(* Schneider Machine Expert - Basic project Modelo final v1.0, file version 2.5.0.0 *)
(* ProjectInformations: Name=Nuevo proyecto *)

HARDWARE
  Cpu 0: TM221CE24T
  EthernetConfiguration: NetworkName=M221, IpAllocationMode=FixedAddress, IpAddress=0.0.0.0, SubnetMask=0.0.0.0
  SerialLineConfiguration: Baud=Baud19200, Parity=ParityEven, DataBits=DataBits8, StopBits=StopBits1, PhysicalMedium=PhysicalMediumRs485, TransmissionMode=TransmissionModeModbusRtu, SlaveId=1, Addressing=SlaveAddressing
  MastTask: UsePeriodScanMode=false, PeriodScan=100
  FastTask: Period=255
  CpuBehavior: StartingMode=StartAsPreviousState, AutoSaveRamOnEeprom=true, WatchdogPeriod=250

SYMBOLS  (address, symbol, comment, settings)
  %M0         "Escalon frontal izquierdo"
  %M1         "Escalon frontal derecho"
  %M2         "Escalon trasero izquierdo"
  %M3         "Escalon trasero derecho"
  %M4         "Sensor frente izquierdo"
  %M5         "Sensor frente medio"
  %M6         "Sensor frente derecho"
  %M7         "Sensor derecha adelante"
  %M8         "Sensor derecha medio"
  %M9         "Sensor derecha atras"
  %M10        "Sensor trasero derecha"
  %M11        "Sensor trasero medio"
  %M12        "Sensor trasero izquierda"
  %M13        "Sensor izquierda atras"
  %M14        "Sensor izquierda medio"
  %M15        "Sensor izquierda adelante"
  %M40        "Reset gen"
  %S6       SB_TB1S  "Base de tiempo de 1 s generada por un reloj interno"
  %TM0        [Preset=5, Base=OneHundredMilliSeconds]
  %TM1        [Preset=5, Base=OneHundredMilliSeconds]
  %TM2        [Preset=5, Base=OneHundredMilliSeconds]
  %TM3        [Preset=5, Base=OneHundredMilliSeconds]
  %TM4        [Preset=5, Base=OneHundredMilliSeconds]
  %TM5        [Preset=5, Base=OneHundredMilliSeconds]
  %TM6        [Preset=5, Base=OneHundredMilliSeconds]
  %TM7        [Preset=5, Base=OneHundredMilliSeconds]
  %TM8        [Preset=5, Base=OneHundredMilliSeconds]
  %TM9        [Preset=5, Base=OneHundredMilliSeconds]
  %TM10       [Preset=5, Base=OneHundredMilliSeconds]
  %TM11       [Preset=5, Base=OneHundredMilliSeconds]
  %TM12       [Preset=5, Base=OneHundredMilliSeconds]
  %TM13       [Preset=5, Base=OneHundredMilliSeconds]
  %TM14       [Preset=5, Base=OneHundredMilliSeconds]
  %TM15       [Preset=5, Base=OneHundredMilliSeconds]
  %C0         [Preset=17]
  %I0.0     ENC1A  "Input"
  %I0.1     ENC1B  "Enable"
  %I0.6     ENC2A
  %I0.7     ENC2B
  %I0.8     MUX  "Data de mux sensores"
  %Q0.4     S0
  %Q0.5     S1
  %Q0.6     S2
  %Q0.7     S3

POU Demux
  (* SectionNumber=1 *)

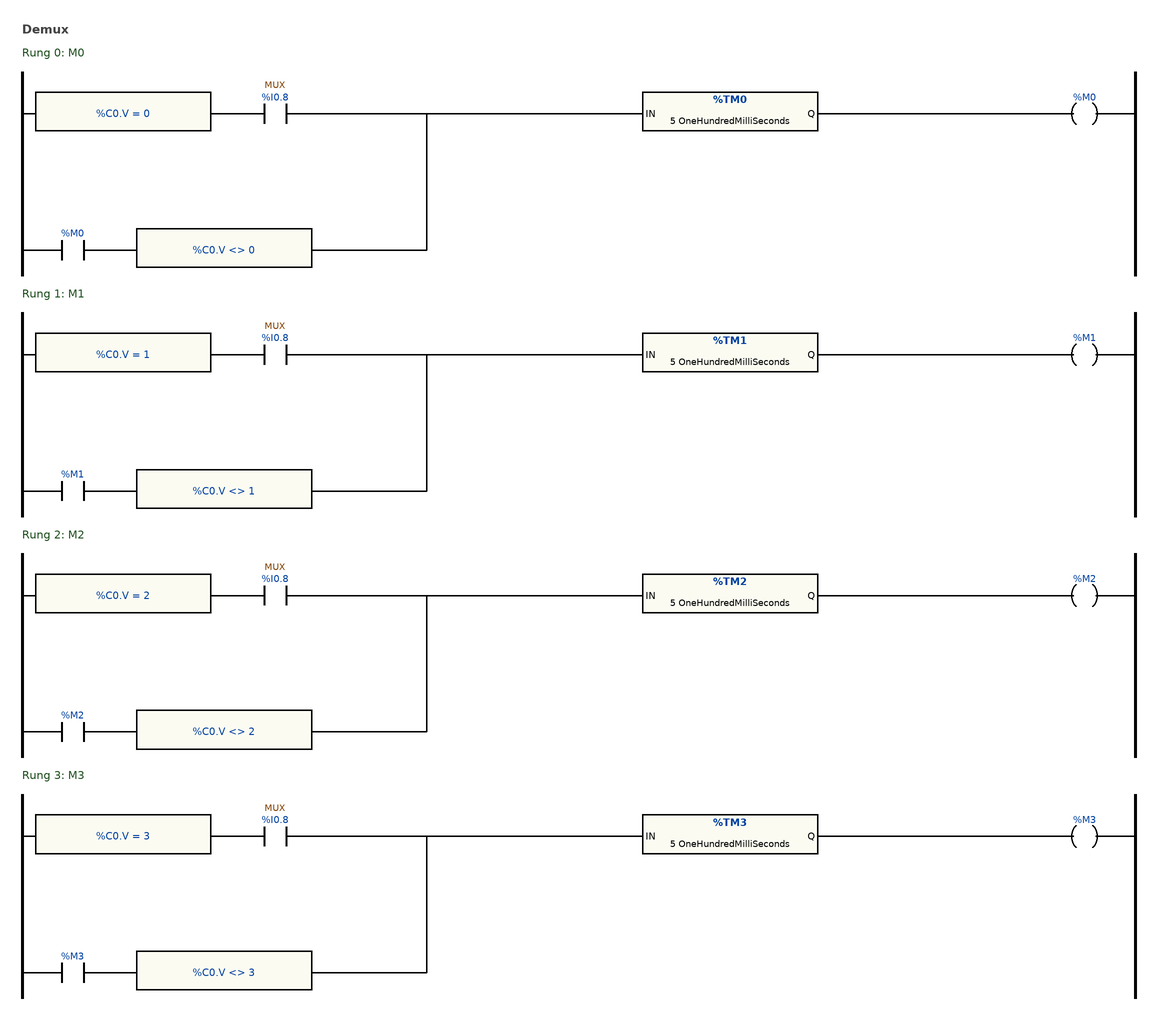

// Rung 0: M0
  BLK %TM0
  LD [ %C0.V = 0 ]
  AND %I0.8               (* MUX *)
  OR( %M0
  AND [ %C0.V <> 0 ]
  )
  IN
  OUT_BLK
  LD Q
  ST %M0
  END_BLK
  // as ST:
  //   %TM0(IN := %C0.V = 0 AND MUX OR %M0 AND %C0.V <> 0);
  //   %M0 := %TM0.Q;

// Rung 1: M1
  BLK %TM1
  LD [ %C0.V = 1 ]
  AND %I0.8               (* MUX *)
  OR( %M1
  AND [ %C0.V <> 1 ]
  )
  IN
  OUT_BLK
  LD Q
  ST %M1
  END_BLK
  // as ST:
  //   %TM1(IN := %C0.V = 1 AND MUX OR %M1 AND %C0.V <> 1);
  //   %M1 := %TM1.Q;

// Rung 2: M2
  BLK %TM2
  LD [ %C0.V = 2 ]
  AND %I0.8               (* MUX *)
  OR( %M2
  AND [ %C0.V <> 2 ]
  )
  IN
  OUT_BLK
  LD Q
  ST %M2
  END_BLK
  // as ST:
  //   %TM2(IN := %C0.V = 2 AND MUX OR %M2 AND %C0.V <> 2);
  //   %M2 := %TM2.Q;

// Rung 3: M3
  BLK %TM3
  LD [ %C0.V = 3 ]
  AND %I0.8               (* MUX *)
  OR( %M3
  AND [ %C0.V <> 3 ]
  )
  IN
  OUT_BLK
  LD Q
  ST %M3
  END_BLK
  // as ST:
  //   %TM3(IN := %C0.V = 3 AND MUX OR %M3 AND %C0.V <> 3);
  //   %M3 := %TM3.Q;

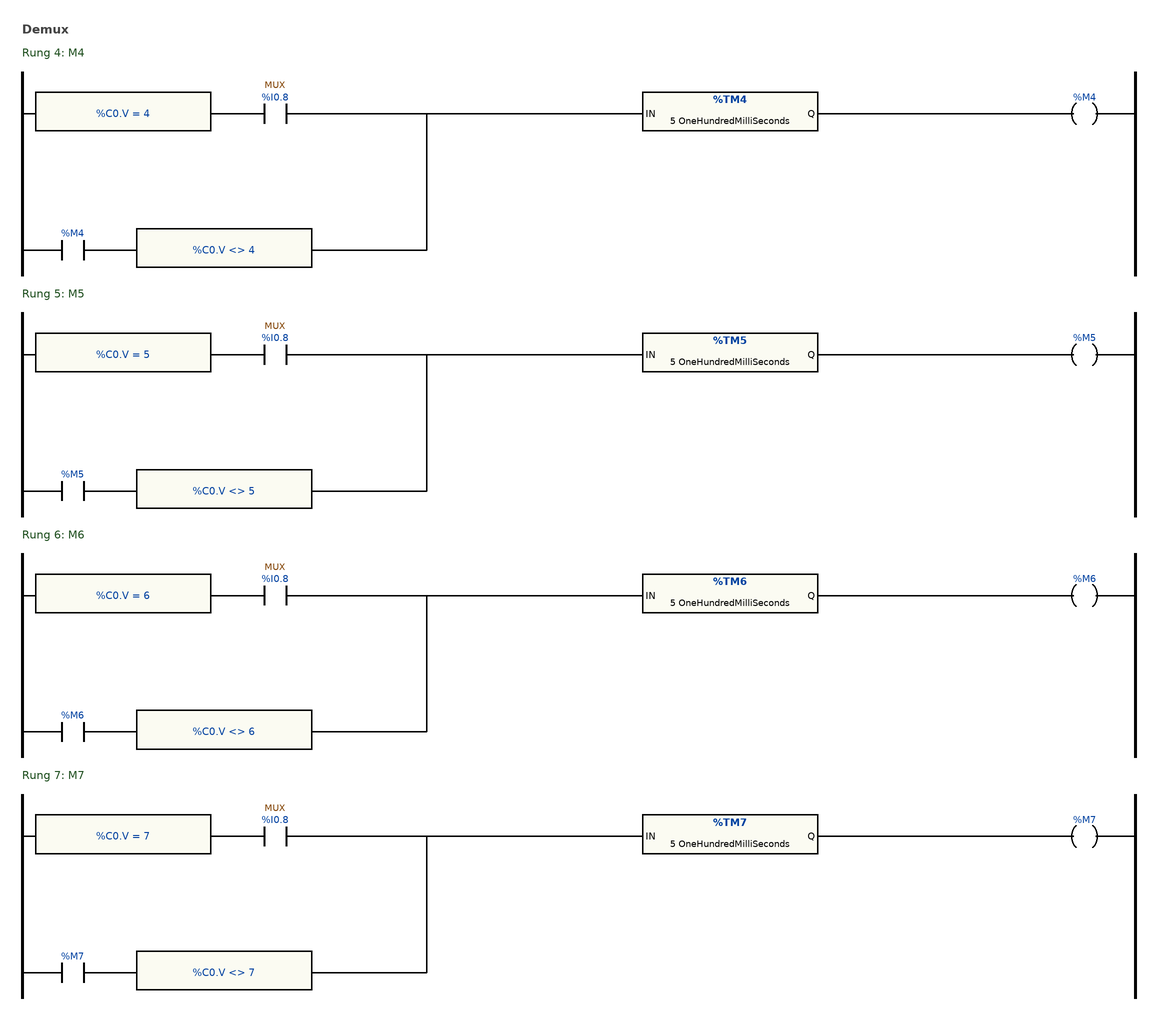

// Rung 4: M4
  BLK %TM4
  LD [ %C0.V = 4 ]
  AND %I0.8               (* MUX *)
  OR( %M4
  AND [ %C0.V <> 4 ]
  )
  IN
  OUT_BLK
  LD Q
  ST %M4
  END_BLK
  // as ST:
  //   %TM4(IN := %C0.V = 4 AND MUX OR %M4 AND %C0.V <> 4);
  //   %M4 := %TM4.Q;

// Rung 5: M5
  BLK %TM5
  LD [ %C0.V = 5 ]
  AND %I0.8               (* MUX *)
  OR( %M5
  AND [ %C0.V <> 5 ]
  )
  IN
  OUT_BLK
  LD Q
  ST %M5
  END_BLK
  // as ST:
  //   %TM5(IN := %C0.V = 5 AND MUX OR %M5 AND %C0.V <> 5);
  //   %M5 := %TM5.Q;

// Rung 6: M6
  BLK %TM6
  LD [ %C0.V = 6 ]
  AND %I0.8               (* MUX *)
  OR( %M6
  AND [ %C0.V <> 6 ]
  )
  IN
  OUT_BLK
  LD Q
  ST %M6
  END_BLK
  // as ST:
  //   %TM6(IN := %C0.V = 6 AND MUX OR %M6 AND %C0.V <> 6);
  //   %M6 := %TM6.Q;

// Rung 7: M7
  BLK %TM7
  LD [ %C0.V = 7 ]
  AND %I0.8               (* MUX *)
  OR( %M7
  AND [ %C0.V <> 7 ]
  )
  IN
  OUT_BLK
  LD Q
  ST %M7
  END_BLK
  // as ST:
  //   %TM7(IN := %C0.V = 7 AND MUX OR %M7 AND %C0.V <> 7);
  //   %M7 := %TM7.Q;

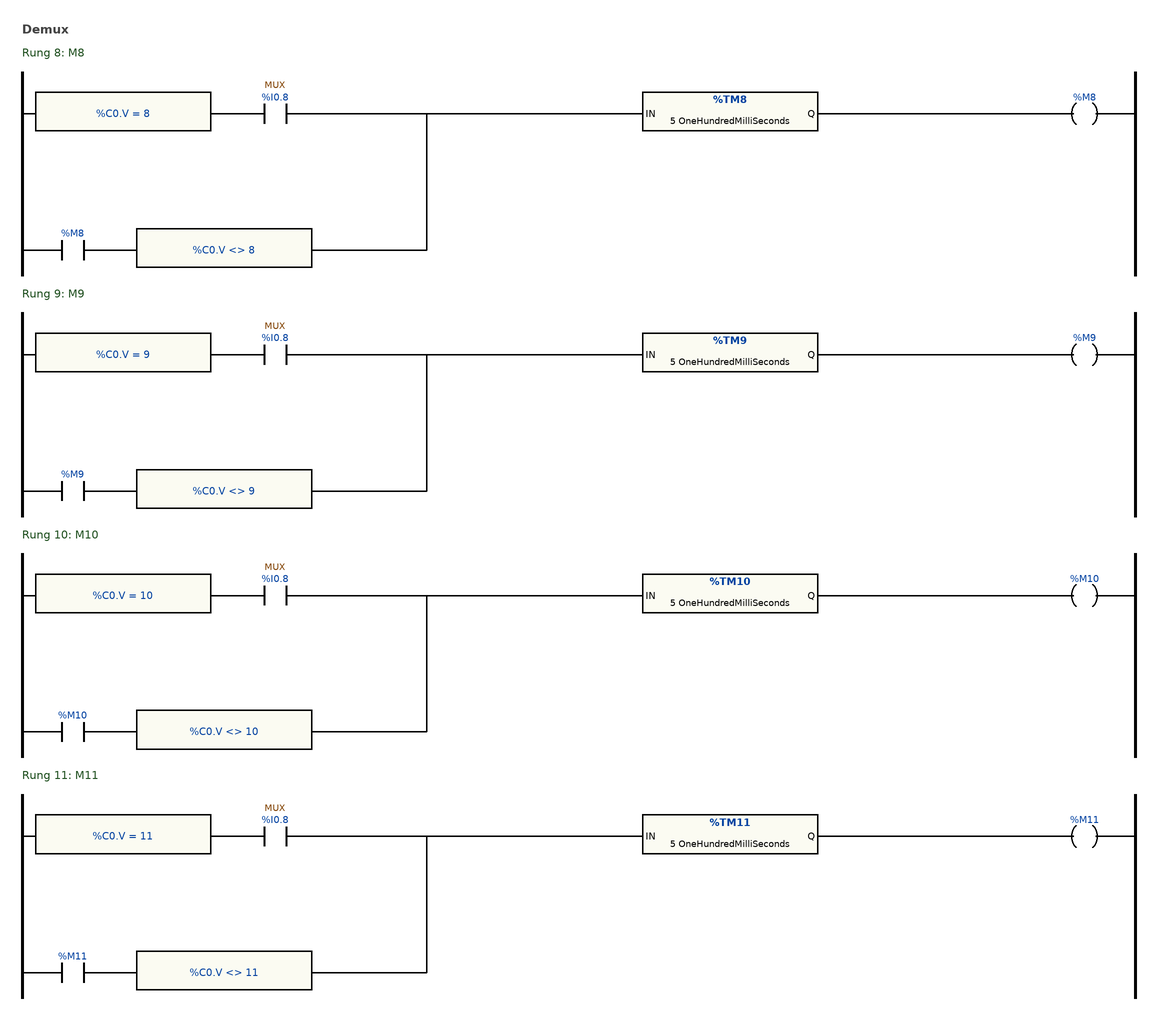

// Rung 8: M8
  BLK %TM8
  LD [ %C0.V = 8 ]
  AND %I0.8               (* MUX *)
  OR( %M8
  AND [ %C0.V <> 8 ]
  )
  IN
  OUT_BLK
  LD Q
  ST %M8
  END_BLK
  // as ST:
  //   %TM8(IN := %C0.V = 8 AND MUX OR %M8 AND %C0.V <> 8);
  //   %M8 := %TM8.Q;

// Rung 9: M9
  BLK %TM9
  LD [ %C0.V = 9 ]
  AND %I0.8               (* MUX *)
  OR( %M9
  AND [ %C0.V <> 9 ]
  )
  IN
  OUT_BLK
  LD Q
  ST %M9
  END_BLK
  // as ST:
  //   %TM9(IN := %C0.V = 9 AND MUX OR %M9 AND %C0.V <> 9);
  //   %M9 := %TM9.Q;

// Rung 10: M10
  BLK %TM10
  LD [ %C0.V = 10 ]
  AND %I0.8               (* MUX *)
  OR( %M10
  AND [ %C0.V <> 10 ]
  )
  IN
  OUT_BLK
  LD Q
  ST %M10
  END_BLK
  // as ST:
  //   %TM10(IN := %C0.V = 10 AND MUX OR %M10 AND %C0.V <> 10);
  //   %M10 := %TM10.Q;

// Rung 11: M11
  BLK %TM11
  LD [ %C0.V = 11 ]
  AND %I0.8               (* MUX *)
  OR( %M11
  AND [ %C0.V <> 11 ]
  )
  IN
  OUT_BLK
  LD Q
  ST %M11
  END_BLK
  // as ST:
  //   %TM11(IN := %C0.V = 11 AND MUX OR %M11 AND %C0.V <> 11);
  //   %M11 := %TM11.Q;

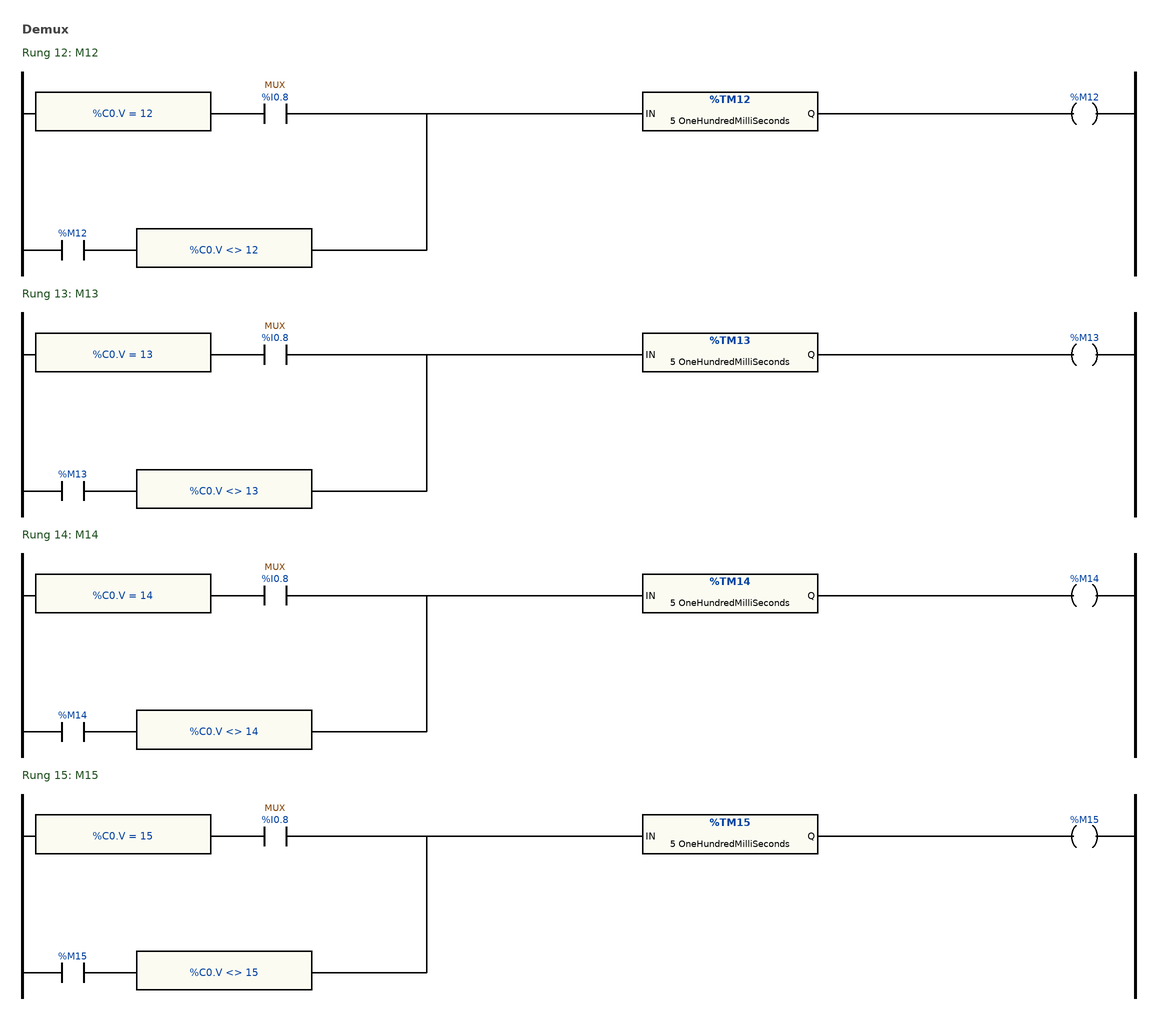

// Rung 12: M12
  BLK %TM12
  LD [ %C0.V = 12 ]
  AND %I0.8               (* MUX *)
  OR( %M12
  AND [ %C0.V <> 12 ]
  )
  IN
  OUT_BLK
  LD Q
  ST %M12
  END_BLK
  // as ST:
  //   %TM12(IN := %C0.V = 12 AND MUX OR %M12 AND %C0.V <> 12);
  //   %M12 := %TM12.Q;

// Rung 13: M13
  BLK %TM13
  LD [ %C0.V = 13 ]
  AND %I0.8               (* MUX *)
  OR( %M13
  AND [ %C0.V <> 13 ]
  )
  IN
  OUT_BLK
  LD Q
  ST %M13
  END_BLK
  // as ST:
  //   %TM13(IN := %C0.V = 13 AND MUX OR %M13 AND %C0.V <> 13);
  //   %M13 := %TM13.Q;

// Rung 14: M14
  BLK %TM14
  LD [ %C0.V = 14 ]
  AND %I0.8               (* MUX *)
  OR( %M14
  AND [ %C0.V <> 14 ]
  )
  IN
  OUT_BLK
  LD Q
  ST %M14
  END_BLK
  // as ST:
  //   %TM14(IN := %C0.V = 14 AND MUX OR %M14 AND %C0.V <> 14);
  //   %M14 := %TM14.Q;

// Rung 15: M15
  BLK %TM15
  LD [ %C0.V = 15 ]
  AND %I0.8               (* MUX *)
  OR( %M15
  AND [ %C0.V <> 15 ]
  )
  IN
  OUT_BLK
  LD Q
  ST %M15
  END_BLK
  // as ST:
  //   %TM15(IN := %C0.V = 15 AND MUX OR %M15 AND %C0.V <> 15);
  //   %M15 := %TM15.Q;

POU Generacion Sx
  (* SectionNumber=2 *)

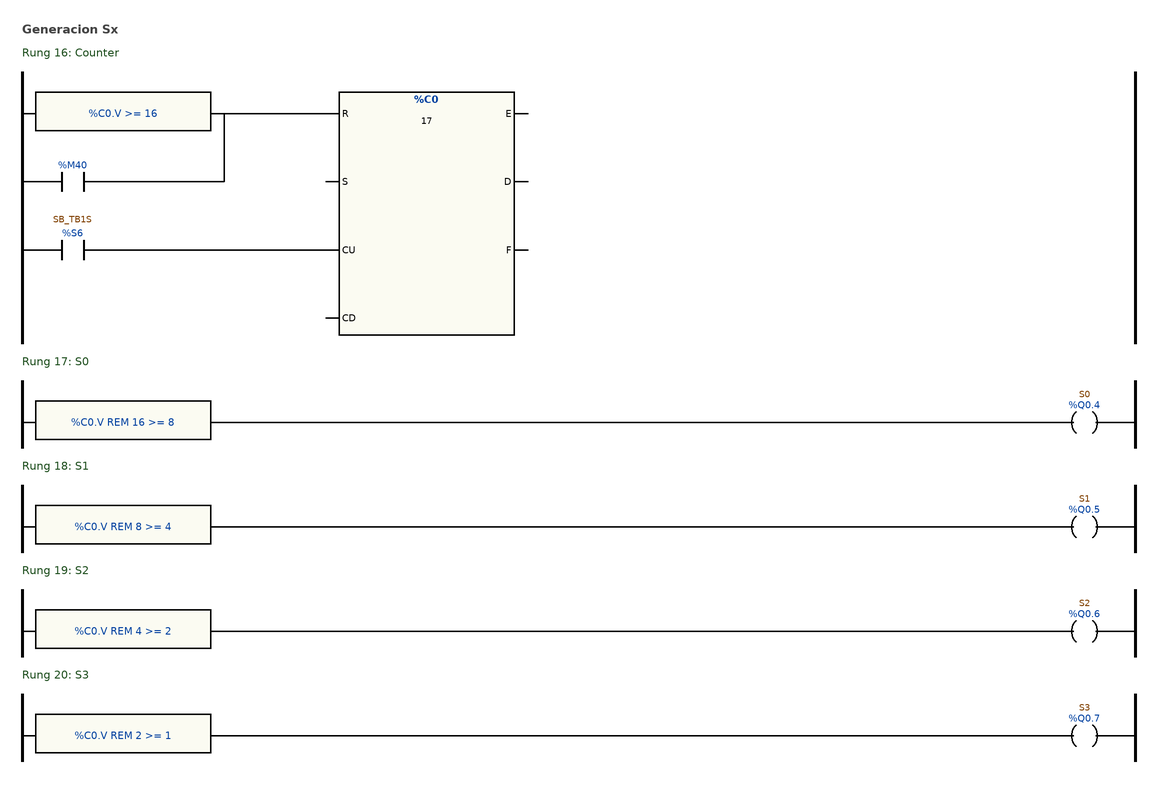

// Rung 16: Counter
  BLK %C0
  LD [ %C0.V >= 16 ]
  OR %M40
  R
  LD %S6                  (* SB_TB1S *)
  CU
  END_BLK
  // as ST:
  //   %C0(R := %C0.V >= 16 OR %M40, CU := SB_TB1S);

// Rung 17: S0
  LD 1
  AND [ %C0.V REM 16 >= 8 ]
  ST %Q0.4                (* S0 *)
  // as ST:
  //   S0 := %C0.V REM 16 >= 8;

// Rung 18: S1
  LD 1
  AND [ %C0.V REM 8 >= 4 ]
  ST %Q0.5                (* S1 *)
  // as ST:
  //   S1 := %C0.V REM 8 >= 4;

// Rung 19: S2
  LD 1
  AND [ %C0.V REM 4 >= 2 ]
  ST %Q0.6                (* S2 *)
  // as ST:
  //   S2 := %C0.V REM 4 >= 2;

// Rung 20: S3
  LD 1
  AND [ %C0.V REM 2 >= 1 ]
  ST %Q0.7                (* S3 *)
  // as ST:
  //   S3 := %C0.V REM 2 >= 1;
